Yaskawa INFORM job: TIR-CORRECTION-BACK-ST-1.JBI

/JOB
//NAME TIR-CORRECTION-BACK-ST-1
//POS
///NPOS 0,0,0,1,0,0
///USER 10
///TOOL 0
///POSTYPE USER
///RECTAN
///RCONF 0,0,0,0,0,0,0,0,0,0,0,0,0,0,0,0,0,0,0,0,0,0,0,0
P00049=2.600,0.000,0.000,0.0000,0.0000,0.0000
//INST
///DATE 2018/11/20 12:44
///ATTR SC,RW
///LVARS 0,0,1,0,0,0,0,0
NOP
'***** get shift value
SUB P049 P049
SET LD000 D030
MUL LD000 100
SETE P049 (1) LD000
'***** F........ sensors
IFTHEN D005=4
	 CALL JOB:TIR-CORR-F-SENSORS-BACK-ST1
ENDIF
END
